INTERFACE I_GraphSettings

METHOD PUBLIC GetLinkByIndex : I_LinkSettings
VAR_INPUT
	Index : UDINT;
END_VAR
END_METHOD

METHOD PUBLIC GetNodeById : I_NodeSettings
VAR_INPUT
	Id : NodeId;
END_VAR
END_METHOD

METHOD PUBLIC GetNodeByIndex : I_NodeSettings
VAR_INPUT
	Index : UDINT;
END_VAR
END_METHOD

PROPERTY PUBLIC HasLinks : Bool
GET
END_GET
END_PROPERTY

PROPERTY PUBLIC HasNodes : Bool
GET
END_GET
END_PROPERTY

PROPERTY PUBLIC LastLinkId : T_MAXSTRING
GET
END_GET
END_PROPERTY

PROPERTY PUBLIC LastNodeId : NodeId
GET
END_GET
END_PROPERTY

PROPERTY PUBLIC LinkCount : UDINT
GET
END_GET
END_PROPERTY

PROPERTY PUBLIC NodeCount : UDINT
GET
END_GET
END_PROPERTY

PROPERTY PUBLIC Uuid : Uuid
GET
END_GET
END_PROPERTY

END_INTERFACE

(* stored: Version 1.1.0.1, ProductVersion 3.1.4024.12
   Itf I_GraphSettings: Id {b57bc97a-963e-05c1-0f33-3eb7c9a4dd29}
   Method GetLinkByIndex: Id {ee8f4ae2-3652-01a5-3721-78fc39870938}
   Method GetNodeById: Id {4ce0beb4-6ffd-0562-17e0-7ed68d51809d}
   Method GetNodeByIndex: Id {7a91d577-fb23-04e1-03d8-b9b8a017606d}
   Property HasLinks: Id {591de848-aba1-00ac-2986-08c9dea1ea35}
   Get Get: Id {b642e848-49ab-00d4-1858-b40246b1d1c3}
   Property HasNodes: Id {67a52646-b6dd-0af9-1915-4f4440357b01}
   Get Get: Id {dc966d73-2bd2-01d0-11a7-9e83bf73aafc}
   Property LastLinkId: Id {238325c8-df9d-0d53-0cb5-795c8f8334de}
   Get Get: Id {f9a5442f-d80b-0010-2e04-59817eb4b5de}
   Property LastNodeId: Id {7060ccda-e72c-052d-357c-e6c341292e76}
   Get Get: Id {1c23985d-cb1c-0683-2c14-9726adbf4b2b}
   Property LinkCount: Id {a29a328d-b738-07f4-19f2-ee435034134e}
   Get Get: Id {6d9cae0d-5d9d-0197-2134-aa76b72a20a4}
   Property NodeCount: Id {3bd3072a-bb37-0231-232b-e2005dd8768c}
   Get Get: Id {6e083d0f-801e-0fec-04e5-4ede63d97fa7}
   Property Uuid: Id {a3cc3d8a-d22c-04e3-0baf-a1bae66d1679}
   Get Get: Id {bccabe69-15ec-01b5-211a-863bf5934827} *)
